// TIA Portal V17 export
// export: Created 2022-07-20T06:59:46.417158Z, ExportSetting WithDefaults, DisplayName Totally Integrated Automation Portal, DisplayVersion V17, DisplayName TIA Portal Openness, DisplayVersion V17, DisplayName TIA Portal Version Control Interface, DisplayVersion V17, DisplayName SINAMICS Startdrive Advanced, DisplayVersion V17, DisplayName SINAMICS Startdrive G130, G150, S120, S150, SINAMICS MV, S210, DisplayVersion V17, DisplayName SINAMICS Startdrive G110M, G120, G120C, G120D, G120P, G115D, DisplayVersion V17, DisplayName STEP 7 Professional, DisplayVersion V17, DisplayName STEP 7 Safety, DisplayVersion V17, DisplayName WinCC Advanced, DisplayVersion V17
FUNCTION_BLOCK "FB10094_GefranIrDryerManager"   // FB10094, LAD
{ S7_Optimized_Access := 'TRUE' }
VERSION : 0.1
// stored: AutoNumber false, IsIECCheckEnabled false, IsRetainMemResEnabled false, MemoryReserve 100, SetENOAutomatically false, UDAEnableTagReadback false
   VAR_INPUT
      IrDryer_Disable : Bool;
      RequestAcknowledge : Bool;
      GefranIrDryerCommunicationIn : "stGefranModuleComIn";
      IrDryer_PowerOnTheBay : Bool;
      IrDryer_ThermalFuse : Bool;
      IrDryer_SetPoint : Real;
      AirPressure_RequestActiveBlowingFan : Bool;
      AirPressure_RequestActiveSuccionFan : Bool;
      AirPressure_Switch : Bool;
   END_VAR
   VAR_OUTPUT
      GefranIrDryerCommunicationOut : "stGefranModuleComOut";
      IrDryer_Disabled : Bool;
      IrDryer_Activated : Bool;
      IrDryer_HeatingInProgress : Bool;
      IrDryer_HeatingDone : Bool;
      IrDryer_ShutdownInProgress : Bool;
      IrDryer_ShutdownTime : Time;
      IrDryer_ShutdownDone : Bool;
      IrDryer_InError : Bool;
      IrDryer_ErrorCode : ULInt;
      AirPressure_ActiveBlowingFan : Bool;
      AirPressure_ActiveSuccionFan : Bool;
      AirPressure_InError : Bool;
   END_VAR
   VAR_IN_OUT
      IrDryer_RequestActiveIrDryer : Bool;
      IrDryer_RequestShutdown : Bool;
   END_VAR
   VAR
      AirExtractorManagementStateDiagram : Int;
      R_TRIG_IrDryerDisable : R_TRIG;
      R_TRIG_RequestActiveIrDryer : R_TRIG;
      R_TRIG_RequestShutdown { S7_SetPoint := 'True'} : R_TRIG;
      R_TRIG_InDryerInError { S7_SetPoint := 'True'} : R_TRIG;
      F_TRIG_RequestActiveIrDryer : F_TRIG;
      F_TRIG_PowerOnBay { S7_SetPoint := 'True'} : F_TRIG;
      TON_IrDryerExtinctionTime { S7_SetPoint := 'True'} : TON_TIME;
      TON_IrErrorDuration { S7_SetPoint := 'True'} : TON_TIME;
   END_VAR
   VAR CONSTANT
      WAIT_FOR_AIR_EXTRACTOR_REQUEST : Int := 0;
      ACTIVE_AIR_EXTRACTOR : Int := 10;
      SHUTDOWN_AIR_EXTRACTOR_IN_PROGRESS : Int := 20;
      REQUEST_DONE : Int := 40;
   END_VAR
BEGIN

REGION Network 1 (SCL): First Scan
   IF "FirstScan" THEN
       ;
   END_IF;
END_REGION

REGION Network 2 (SCL): Edge Signals & Timers
   REGION EDGE SIGNALS
       #R_TRIG_RequestActiveIrDryer(CLK := #IrDryer_RequestActiveIrDryer);
       #R_TRIG_RequestShutdown(CLK := #IrDryer_RequestShutdown);
       #R_TRIG_InDryerInError(CLK := #IrDryer_InError);
       #R_TRIG_IrDryerDisable(CLK := #IrDryer_Disable);

       #F_TRIG_RequestActiveIrDryer(CLK := #IrDryer_RequestActiveIrDryer);
       #F_TRIG_PowerOnBay(CLK := #IrDryer_PowerOnTheBay);
   END_REGION

   REGION TIMERS
       #TON_IrDryerExtinctionTime(IN := #IrDryer_ShutdownInProgress AND #IrDryer_PowerOnTheBay,
                                  PT := T#5m,
                                  ET => #IrDryer_ShutdownTime);
       #TON_IrErrorDuration(IN := #IrDryer_ErrorCode <> 0,
                            PT := T#5s);
   END_REGION
END_REGION

REGION Network 3 (SCL): Ir Dryer Commands Management
   IF #F_TRIG_PowerOnBay.Q OR #R_TRIG_InDryerInError.Q OR #IrDryer_Disable OR #IrDryer_ShutdownInProgress THEN
       #IrDryer_RequestActiveIrDryer := FALSE;
   END_IF;
END_REGION

REGION Network 4 (SCL): Ir Dryer Lamps Management
   IF NOT(#IrDryer_Disable) THEN //Active Lamps
       IF #IrDryer_RequestActiveIrDryer AND NOT (#IrDryer_RequestShutdown) THEN
           #GefranIrDryerCommunicationOut.Module[0].Status_RW_305.Auto_Manual := TRUE;
           #GefranIrDryerCommunicationOut.Module[0].Status_RW_305.ON_OFF := FALSE;
       ELSE
           #GefranIrDryerCommunicationOut.Module[0].Status_RW_305.Auto_Manual := FALSE;
           #GefranIrDryerCommunicationOut.Module[0].Status_RW_305.ON_OFF := TRUE;
       END_IF;

       //Set Point Management
       #GefranIrDryerCommunicationOut.Module[0].Manual_Power := #IrDryer_SetPoint;
       #GefranIrDryerCommunicationOut.Module[1].Manual_Power := #IrDryer_SetPoint;
       #GefranIrDryerCommunicationOut.Module[2].Manual_Power := #IrDryer_SetPoint;
       #GefranIrDryerCommunicationOut.Module[3].Manual_Power := #IrDryer_SetPoint;
   ELSE
       #GefranIrDryerCommunicationOut.Module[0].Status_RW_305.Auto_Manual := FALSE;
       #GefranIrDryerCommunicationOut.Module[0].Status_RW_305.ON_OFF := TRUE;

       #GefranIrDryerCommunicationOut.Module[0].Manual_Power := 0;
       #GefranIrDryerCommunicationOut.Module[1].Manual_Power := 0;
       #GefranIrDryerCommunicationOut.Module[2].Manual_Power := 0;
       #GefranIrDryerCommunicationOut.Module[3].Manual_Power := 0;
   END_IF;
END_REGION

REGION Network 5 (SCL): Ir Dryer Air Pressure Management
   IF #R_TRIG_RequestActiveIrDryer.Q AND NOT (#IrDryer_Disable) THEN
       #IrDryer_ShutdownDone := FALSE;
       #AirExtractorManagementStateDiagram := #ACTIVE_AIR_EXTRACTOR;
   ELSIF
       (#R_TRIG_RequestShutdown.Q AND NOT (#IrDryer_Disabled)) OR
       (#F_TRIG_RequestActiveIrDryer.Q AND NOT (#IrDryer_Disabled)) OR
       (#R_TRIG_IrDryerDisable.Q AND (#AirExtractorManagementStateDiagram = #ACTIVE_AIR_EXTRACTOR))
   THEN
       #AirExtractorManagementStateDiagram := #SHUTDOWN_AIR_EXTRACTOR_IN_PROGRESS;
   END_IF;

   CASE #AirExtractorManagementStateDiagram OF
       #WAIT_FOR_AIR_EXTRACTOR_REQUEST:
           #AirPressure_ActiveSuccionFan := FALSE;
           #AirPressure_ActiveBlowingFan := FALSE;

       #ACTIVE_AIR_EXTRACTOR:
           #AirPressure_ActiveSuccionFan := TRUE;
           #AirPressure_ActiveBlowingFan := TRUE;

           IF #R_TRIG_RequestShutdown.Q OR #F_TRIG_RequestActiveIrDryer.Q THEN
               #AirExtractorManagementStateDiagram := #SHUTDOWN_AIR_EXTRACTOR_IN_PROGRESS;
           END_IF;
       #SHUTDOWN_AIR_EXTRACTOR_IN_PROGRESS:
           #AirPressure_ActiveSuccionFan := TRUE;
           #AirPressure_ActiveBlowingFan := TRUE;

           IF #TON_IrDryerExtinctionTime.Q THEN
               #AirPressure_ActiveSuccionFan := FALSE;
               #AirPressure_ActiveBlowingFan := FALSE;
               #IrDryer_ShutdownInProgress := FALSE;
               #IrDryer_ShutdownDone := TRUE;
               #AirExtractorManagementStateDiagram := #REQUEST_DONE;
           END_IF;
       #REQUEST_DONE:
           #AirPressure_ActiveSuccionFan := FALSE;
           #AirPressure_ActiveBlowingFan := FALSE;
           #AirExtractorManagementStateDiagram := #WAIT_FOR_AIR_EXTRACTOR_REQUEST;
   END_CASE;
END_REGION

REGION Network 6 (SCL): Ir Dryer States Management
   #IrDryer_Activated := #GefranIrDryerCommunicationIn.Module[0].StatusW_RO_463.Auto_Manual AND NOT (#GefranIrDryerCommunicationIn.Module[0].StatusW_RO_463.ON_OFF);

   #IrDryer_HeatingInProgress := #GefranIrDryerCommunicationIn.Module[0].Status4_634.Phase_SoftstartActive OR (#IrDryer_Activated AND #GefranIrDryerCommunicationIn.Module[0].Load.Output_Control_Value <> #IrDryer_SetPoint);

   #IrDryer_HeatingDone := #GefranIrDryerCommunicationIn.Module[0].Status4_634.Phase_SoftstartEnd AND #GefranIrDryerCommunicationIn.Module[0].Load.Output_Control_Value = #IrDryer_SetPoint;

   #IrDryer_Disabled := #IrDryer_Disable AND
   (NOT (#GefranIrDryerCommunicationOut.Module[0].Status_RW_305.Auto_Manual) AND #GefranIrDryerCommunicationOut.Module[0].Status_RW_305.ON_OFF) AND
   (#GefranIrDryerCommunicationOut.Module[0].Manual_Power = 0 AND #GefranIrDryerCommunicationOut.Module[1].Manual_Power = 0 AND #GefranIrDryerCommunicationOut.Module[2].Manual_Power = 0 AND #GefranIrDryerCommunicationOut.Module[3].Manual_Power = 0) AND
   NOT (#AirPressure_ActiveSuccionFan) AND NOT (#AirPressure_ActiveBlowingFan);

   #IrDryer_ShutdownInProgress := #AirExtractorManagementStateDiagram = #SHUTDOWN_AIR_EXTRACTOR_IN_PROGRESS;

   IF #TON_IrDryerExtinctionTime.Q THEN
       #IrDryer_ShutdownDone := TRUE;
   ELSIF #TON_IrDryerExtinctionTime.ET > T#0s THEN
       #IrDryer_ShutdownDone := FALSE;
   END_IF;
END_REGION

REGION Network 7 (SCL): Ir Dryer Error Managament
   //Air Switch Error Management
   IF #IrDryer_Activated AND #IrDryer_HeatingDone AND NOT #AirPressure_Switch THEN
       #AirPressure_InError := TRUE;
   END_IF;

   //Ir Dryer Lamps Error 
   IF #TON_IrErrorDuration.Q THEN
       #IrDryer_InError := TRUE;
   END_IF;

   #IrDryer_ErrorCode.%X0 := (NOT (#IrDryer_ThermalFuse) AND #IrDryer_RequestActiveIrDryer) OR #IrDryer_ErrorCode.%X0;

   #IrDryer_ErrorCode.%X1 := #GefranIrDryerCommunicationIn.Module[0].Status4_634.Temperature_Sensor_Broken OR #IrDryer_ErrorCode.%X1;
   #IrDryer_ErrorCode.%X2 := #GefranIrDryerCommunicationIn.Module[0].Status4_634.OverHeat OR #IrDryer_ErrorCode.%X2;
   #IrDryer_ErrorCode.%X3 := #GefranIrDryerCommunicationIn.Module[0].Status4_634.Frequency_Error OR #IrDryer_ErrorCode.%X3;
   #IrDryer_ErrorCode.%X4 := #GefranIrDryerCommunicationIn.Module[0].Status4_634."60Hz" OR #IrDryer_ErrorCode.%X4;
   #IrDryer_ErrorCode.%X5 := #GefranIrDryerCommunicationIn.Module[0].Status4_634.Short_Circuit_Current OR #IrDryer_ErrorCode.%X5;
   #IrDryer_ErrorCode.%X6 := #GefranIrDryerCommunicationIn.Module[0].Status4_634.Over_Peak_Current OR #IrDryer_ErrorCode.%X6;
   #IrDryer_ErrorCode.%X7 := #GefranIrDryerCommunicationIn.Module[0].Status4_634.Over_RMS_Current OR #IrDryer_ErrorCode.%X7;
   #IrDryer_ErrorCode.%X8 := #GefranIrDryerCommunicationIn.Module[0].Status4_634.Alpower_Or_HWoverheat OR #IrDryer_ErrorCode.%X8;
   #IrDryer_ErrorCode.%X9 := #GefranIrDryerCommunicationIn.Module[0].Status4_634.Fuse_open OR #IrDryer_ErrorCode.%X9;

   #IrDryer_ErrorCode.%X10 := #GefranIrDryerCommunicationIn.Module[1].Status4_634.Temperature_Sensor_Broken OR #IrDryer_ErrorCode.%X10;
   #IrDryer_ErrorCode.%X11 := #GefranIrDryerCommunicationIn.Module[1].Status4_634.OverHeat OR #IrDryer_ErrorCode.%X11;
   #IrDryer_ErrorCode.%X12 := #GefranIrDryerCommunicationIn.Module[1].Status4_634.Frequency_Error OR #IrDryer_ErrorCode.%X12;
   #IrDryer_ErrorCode.%X13 := #GefranIrDryerCommunicationIn.Module[1].Status4_634."60Hz" OR #IrDryer_ErrorCode.%X13;
   #IrDryer_ErrorCode.%X14 := #GefranIrDryerCommunicationIn.Module[1].Status4_634.Short_Circuit_Current OR #IrDryer_ErrorCode.%X14;
   #IrDryer_ErrorCode.%X15 := #GefranIrDryerCommunicationIn.Module[1].Status4_634.Over_Peak_Current OR #IrDryer_ErrorCode.%X15;
   #IrDryer_ErrorCode.%X16 := #GefranIrDryerCommunicationIn.Module[1].Status4_634.Over_RMS_Current OR #IrDryer_ErrorCode.%X16;
   #IrDryer_ErrorCode.%X17 := #GefranIrDryerCommunicationIn.Module[1].Status4_634.Alpower_Or_HWoverheat OR #IrDryer_ErrorCode.%X17;
   #IrDryer_ErrorCode.%X18 := #GefranIrDryerCommunicationIn.Module[1].Status4_634.Fuse_open OR #IrDryer_ErrorCode.%X18;

   #IrDryer_ErrorCode.%X19 := #GefranIrDryerCommunicationIn.Module[2].Status4_634.Temperature_Sensor_Broken OR #IrDryer_ErrorCode.%X19;
   #IrDryer_ErrorCode.%X20 := #GefranIrDryerCommunicationIn.Module[2].Status4_634.OverHeat OR #IrDryer_ErrorCode.%X20;
   #IrDryer_ErrorCode.%X21 := #GefranIrDryerCommunicationIn.Module[2].Status4_634.Frequency_Error OR #IrDryer_ErrorCode.%X21;
   #IrDryer_ErrorCode.%X22 := #GefranIrDryerCommunicationIn.Module[2].Status4_634."60Hz" OR #IrDryer_ErrorCode.%X22;
   #IrDryer_ErrorCode.%X23 := #GefranIrDryerCommunicationIn.Module[2].Status4_634.Short_Circuit_Current OR #IrDryer_ErrorCode.%X23;
   #IrDryer_ErrorCode.%X24 := #GefranIrDryerCommunicationIn.Module[2].Status4_634.Over_Peak_Current OR #IrDryer_ErrorCode.%X24;
   #IrDryer_ErrorCode.%X25 := #GefranIrDryerCommunicationIn.Module[2].Status4_634.Over_RMS_Current OR #IrDryer_ErrorCode.%X25;
   #IrDryer_ErrorCode.%X26 := #GefranIrDryerCommunicationIn.Module[2].Status4_634.Alpower_Or_HWoverheat OR #IrDryer_ErrorCode.%X26;
   #IrDryer_ErrorCode.%X27 := #GefranIrDryerCommunicationIn.Module[2].Status4_634.Fuse_open OR #IrDryer_ErrorCode.%X27;

   #IrDryer_ErrorCode.%X28 := #GefranIrDryerCommunicationIn.Module[3].Status4_634.Temperature_Sensor_Broken OR #IrDryer_ErrorCode.%X28;
   #IrDryer_ErrorCode.%X29 := #GefranIrDryerCommunicationIn.Module[3].Status4_634.OverHeat OR #IrDryer_ErrorCode.%X29;
   #IrDryer_ErrorCode.%X30 := #GefranIrDryerCommunicationIn.Module[3].Status4_634.Frequency_Error OR #IrDryer_ErrorCode.%X30;
   #IrDryer_ErrorCode.%X31 := #GefranIrDryerCommunicationIn.Module[3].Status4_634."60Hz" OR #IrDryer_ErrorCode.%X31;
   #IrDryer_ErrorCode.%X32 := #GefranIrDryerCommunicationIn.Module[3].Status4_634.Short_Circuit_Current OR #IrDryer_ErrorCode.%X32;
   #IrDryer_ErrorCode.%X33 := #GefranIrDryerCommunicationIn.Module[3].Status4_634.Over_Peak_Current OR #IrDryer_ErrorCode.%X33;
   #IrDryer_ErrorCode.%X34 := #GefranIrDryerCommunicationIn.Module[3].Status4_634.Over_RMS_Current OR #IrDryer_ErrorCode.%X34;
   #IrDryer_ErrorCode.%X35 := #GefranIrDryerCommunicationIn.Module[3].Status4_634.Alpower_Or_HWoverheat OR #IrDryer_ErrorCode.%X35;
   #IrDryer_ErrorCode.%X36 := #GefranIrDryerCommunicationIn.Module[3].Status4_634.Fuse_open OR #IrDryer_ErrorCode.%X36;

   //Acknwoledge Management
   IF #RequestAcknowledge THEN
       #IrDryer_ErrorCode := 0;
       #AirPressure_InError := FALSE;
       #IrDryer_InError := FALSE;
   END_IF;
END_REGION
END_FUNCTION_BLOCK
